                                        FB_Bacnet.StartStopCommand_143.bEnWrite := TRUE;
                                        FB_Bacnet.StartStopCommand_143.bVal := TRUE;
                                    17: 
                                        
                                        FB_Bacnet.StartStopCommand_144.bEnWrite := TRUE;
                                        FB_Bacnet.StartStopCommand_144.bVal := TRUE;
                                    18: 
                                        
                                        FB_Bacnet.StartStopCommand_145.bEnWrite := TRUE;
                                        FB_Bacnet.StartStopCommand_145.bVal := TRUE;
                                    19: 
                                        
                                        FB_Bacnet.StartStopCommand_146.bEnWrite := TRUE;
                                        FB_Bacnet.StartStopCommand_146.bVal := TRUE;
                                    20: 
                                        
                                        FB_Bacnet.StartStopCommand_147.bEnWrite := TRUE;
                                        FB_Bacnet.StartStopCommand_147.bVal := TRUE;
                                    21: 
                                        
                                        FB_Bacnet.StartStopCommand_148.bEnWrite := TRUE;
                                        FB_Bacnet.StartStopCommand_148.bVal := TRUE;
                                    22: 
                                        
                                        FB_Bacnet.StartStopCommand_149.bEnWrite := TRUE;
                                        FB_Bacnet.StartStopCommand_149.bVal := TRUE;
                                    23: 
                                        
                                        FB_Bacnet.StartStopCommand_176.bEnWrite := TRUE;
                                        FB_Bacnet.StartStopCommand_176.bVal := TRUE;
                                    24: 
                                        
                                        FB_Bacnet.StartStopCommand_241.bEnWrite := TRUE;
                                        FB_Bacnet.StartStopCommand_241.bVal := TRUE;
                                    25: 
                                        
                                        FB_Bacnet.StartStopCommand_226.bEnWrite := TRUE;
                                        FB_Bacnet.StartStopCommand_226.bVal := TRUE;
                                END_CASE
                            END_IF
                        END_FOR
                    END_IF
                    // Schedule Unit OFF
                    IF wSchedWDHourEndF38_ = currH AND wSchedWDMinEndF38_ = currM AND NOT bUnitTriggered THEN
                        bUnitTriggered := TRUE;
                        FOR i := 1 TO 25 DO
                            // Send command unit OFF
                            IF bUnitF38_[i] THEN 
                                CASE i OF
                                    1: 
                                        
                                        FB_Bacnet.StartStopCommand_128.bEnWrite := TRUE;
                                        FB_Bacnet.StartStopCommand_128.bVal := FALSE;
                                    2: 
                                        
                                        FB_Bacnet.StartStopCommand_129.bEnWrite := TRUE;
                                        FB_Bacnet.StartStopCommand_129.bVal := FALSE;
                                    3: 
                                        
                                        FB_Bacnet.StartStopCommand_130.bEnWrite := TRUE;
                                        FB_Bacnet.StartStopCommand_130.bVal := FALSE;
                                    4: 
                                        
                                        FB_Bacnet.StartStopCommand_131.bEnWrite := TRUE;
                                        FB_Bacnet.StartStopCommand_131.bVal := FALSE;
                                    5: 
                                        
                                        FB_Bacnet.StartStopCommand_132.bEnWrite := TRUE;
                                        FB_Bacnet.StartStopCommand_132.bVal := FALSE;
                                    6: 
                                        
                                        FB_Bacnet.StartStopCommand_133.bEnWrite := TRUE;
                                        FB_Bacnet.StartStopCommand_133.bVal := FALSE;
                                    7: 
                                        
                                        FB_Bacnet.StartStopCommand_134.bEnWrite := TRUE;
                                        FB_Bacnet.StartStopCommand_134.bVal := FALSE;
                                    8: 
                                        
                                        FB_Bacnet.StartStopCommand_135.bEnWrite := TRUE;
                                        FB_Bacnet.StartStopCommand_135.bVal := FALSE;
                                    9: 
                                        
                                        FB_Bacnet.StartStopCommand_136.bEnWrite := TRUE;
                                        FB_Bacnet.StartStopCommand_136.bVal := FALSE;
                                    10: 
                                        
                                        FB_Bacnet.StartStopCommand_137.bEnWrite := TRUE;
                                        FB_Bacnet.StartStopCommand_137.bVal := FALSE;
                                    11: 
                                        
                                        FB_Bacnet.StartStopCommand_138.bEnWrite := TRUE;
                                        FB_Bacnet.StartStopCommand_138.bVal := FALSE;
                                    12: 
                                        
                                        FB_Bacnet.StartStopCommand_139.bEnWrite := TRUE;
                                        FB_Bacnet.StartStopCommand_139.bVal := FALSE;
                                    13: 
                                        
                                        FB_Bacnet.StartStopCommand_140.bEnWrite := TRUE;
                                        FB_Bacnet.StartStopCommand_140.bVal := FALSE;
                                    14: 
                                        
                                        FB_Bacnet.StartStopCommand_141.bEnWrite := TRUE;
                                        FB_Bacnet.StartStopCommand_141.bVal := FALSE;
                                    15: 
                                        
                                        FB_Bacnet.StartStopCommand_142.bEnWrite := TRUE;
                                        FB_Bacnet.StartStopCommand_142.bVal := FALSE;
                                    16: 
                                        
                                        FB_Bacnet.StartStopCommand_143.bEnWrite := TRUE;
                                        FB_Bacnet.StartStopCommand_143.bVal := FALSE;
                                    17: 
                                        
                                        FB_Bacnet.StartStopCommand_144.bEnWrite := TRUE;
                                        FB_Bacnet.StartStopCommand_144.bVal := FALSE;
                                    18: 
                                        
                                        FB_Bacnet.StartStopCommand_145.bEnWrite := TRUE;
                                        FB_Bacnet.StartStopCommand_145.bVal := FALSE;
                                    19: 
                                        
                                        FB_Bacnet.StartStopCommand_146.bEnWrite := TRUE;
                                        FB_Bacnet.StartStopCommand_146.bVal := FALSE;
                                    20: 
                                        
                                        FB_Bacnet.StartStopCommand_147.bEnWrite := TRUE;
                                        FB_Bacnet.StartStopCommand_147.bVal := FALSE;
                                    21: 
                                        
                                        FB_Bacnet.StartStopCommand_148.bEnWrite := TRUE;
                                        FB_Bacnet.StartStopCommand_148.bVal := FALSE;
                                    22: 
                                        
                                        FB_Bacnet.StartStopCommand_149.bEnWrite := TRUE;
                                        FB_Bacnet.StartStopCommand_149.bVal := FALSE;
                                    23: 
                                        
                                        FB_Bacnet.StartStopCommand_176.bEnWrite := TRUE;
                                        FB_Bacnet.StartStopCommand_176.bVal := FALSE;
                                    24: 
                                        
                                        FB_Bacnet.StartStopCommand_241.bEnWrite := TRUE;
                                        FB_Bacnet.StartStopCommand_241.bVal := FALSE;
                                    25: 
                                        
                                        FB_Bacnet.StartStopCommand_226.bEnWrite := TRUE;
                                        FB_Bacnet.StartStopCommand_226.bVal := FALSE;
                                END_CASE
                            END_IF
                        END_FOR
                    END_IF
                END_IF
            END_IF
        END_IF

        // Weekend schedule
        IF currD = 0 OR currD = 6 THEN
            IF (wSchedWEHourStartF38_ <> wSchedWEHourEndF38_ OR wSchedWEMinStartF38_ <> wSchedWEMinEndF38_) THEN
                // Schedule Unit ON
                IF wSchedWEHourStartF38_ = currH AND wSchedWEMinStartF38_ = currM AND NOT bUnitTriggered THEN
                    bUnitTriggered := TRUE;
                    FOR i := 1 TO 25 DO
                        // Send command unit ON
                        IF bUnitF38_[i] THEN 
                            CASE i OF
                                1: 
                                    
                                    FB_Bacnet.StartStopCommand_128.bEnWrite := TRUE;
                                    FB_Bacnet.StartStopCommand_128.bVal := TRUE;
                                2: 
                                    
                                    FB_Bacnet.StartStopCommand_129.bEnWrite := TRUE;
                                    FB_Bacnet.StartStopCommand_129.bVal := TRUE;
                                3: 
                                    
                                    FB_Bacnet.StartStopCommand_130.bEnWrite := TRUE;
                                    FB_Bacnet.StartStopCommand_130.bVal := TRUE;
                                4: 
                                    
                                    FB_Bacnet.StartStopCommand_131.bEnWrite := TRUE;
                                    FB_Bacnet.StartStopCommand_131.bVal := TRUE;
                                5: 
                                    
                                    FB_Bacnet.StartStopCommand_132.bEnWrite := TRUE;
                                    FB_Bacnet.StartStopCommand_132.bVal := TRUE;
                                6: 
                                    
                                    FB_Bacnet.StartStopCommand_133.bEnWrite := TRUE;
                                    FB_Bacnet.StartStopCommand_133.bVal := TRUE;
                                7: 
                                    
                                    FB_Bacnet.StartStopCommand_134.bEnWrite := TRUE;
                                    FB_Bacnet.StartStopCommand_134.bVal := TRUE;
                                8: 
                                    
                                    FB_Bacnet.StartStopCommand_135.bEnWrite := TRUE;
                                    FB_Bacnet.StartStopCommand_135.bVal := TRUE;
                                9: 
                                    
                                    FB_Bacnet.StartStopCommand_136.bEnWrite := TRUE;
                                    FB_Bacnet.StartStopCommand_136.bVal := TRUE;
                                10: 
                                    
                                    FB_Bacnet.StartStopCommand_137.bEnWrite := TRUE;
                                    FB_Bacnet.StartStopCommand_137.bVal := TRUE;
                                11: 
                                    
                                    FB_Bacnet.StartStopCommand_138.bEnWrite := TRUE;
                                    FB_Bacnet.StartStopCommand_138.bVal := TRUE;
                                12: 
                                    
                                    FB_Bacnet.StartStopCommand_139.bEnWrite := TRUE;
                                    FB_Bacnet.StartStopCommand_139.bVal := TRUE;
                                13: 
                                    
                                    FB_Bacnet.StartStopCommand_140.bEnWrite := TRUE;
                                    FB_Bacnet.StartStopCommand_140.bVal := TRUE;
                                14: 
                                    
                                    FB_Bacnet.StartStopCommand_141.bEnWrite := TRUE;
                                    FB_Bacnet.StartStopCommand_141.bVal := TRUE;
                                15: 
                                    
                                    FB_Bacnet.StartStopCommand_142.bEnWrite := TRUE;
                                    FB_Bacnet.StartStopCommand_142.bVal := TRUE;
                                16: 
                                    
                                    FB_Bacnet.StartStopCommand_143.bEnWrite := TRUE;
                                    FB_Bacnet.StartStopCommand_143.bVal := TRUE;
                                17: 
                                    
                                    FB_Bacnet.StartStopCommand_144.bEnWrite := TRUE;
                                    FB_Bacnet.StartStopCommand_144.bVal := TRUE;
                                18: 
                                    
                                    FB_Bacnet.StartStopCommand_145.bEnWrite := TRUE;
                                    FB_Bacnet.StartStopCommand_145.bVal := TRUE;
                                19: 
                                    
                                    FB_Bacnet.StartStopCommand_146.bEnWrite := TRUE;
                                    FB_Bacnet.StartStopCommand_146.bVal := TRUE;
                                20: 
                                    
                                    FB_Bacnet.StartStopCommand_147.bEnWrite := TRUE;
                                    FB_Bacnet.StartStopCommand_147.bVal := TRUE;
                                21: 
                                    
                                    FB_Bacnet.StartStopCommand_148.bEnWrite := TRUE;
                                    FB_Bacnet.StartStopCommand_148.bVal := TRUE;
                                22: 
                                    
                                    FB_Bacnet.StartStopCommand_149.bEnWrite := TRUE;
                                    FB_Bacnet.StartStopCommand_149.bVal := TRUE;
                                23: 
                                    
                                    FB_Bacnet.StartStopCommand_176.bEnWrite := TRUE;
                                    FB_Bacnet.StartStopCommand_176.bVal := TRUE;
                                24: 
                                    
                                    FB_Bacnet.StartStopCommand_241.bEnWrite := TRUE;
                                    FB_Bacnet.StartStopCommand_241.bVal := TRUE;
                                25: 
                                    
                                    FB_Bacnet.StartStopCommand_226.bEnWrite := TRUE;
                                    FB_Bacnet.StartStopCommand_226.bVal := TRUE;
                            END_CASE
                        END_IF
                    END_FOR        
                END_IF
                // Schedule Unit OFF
                IF wSchedWEHourEndF38_ = currH AND wSchedWEMinEndF38_ = currM AND NOT bUnitTriggered THEN
                    bUnitTriggered := TRUE;
                    FOR i := 1 TO 25 DO
                        // Send command unit OFF
                        IF bUnitF38_[i] THEN 
                            CASE i OF
                                1: 
                                    
                                    FB_Bacnet.StartStopCommand_128.bEnWrite := TRUE;
                                    FB_Bacnet.StartStopCommand_128.bVal := FALSE;
                                2: 
                                    
                                    FB_Bacnet.StartStopCommand_129.bEnWrite := TRUE;
                                    FB_Bacnet.StartStopCommand_129.bVal := FALSE;
                                3: 
                                    
                                    FB_Bacnet.StartStopCommand_130.bEnWrite := TRUE;
                                    FB_Bacnet.StartStopCommand_130.bVal := FALSE;
                                4: 
                                    
                                    FB_Bacnet.StartStopCommand_131.bEnWrite := TRUE;
                                    FB_Bacnet.StartStopCommand_131.bVal := FALSE;
                                5: 
                                    
                                    FB_Bacnet.StartStopCommand_132.bEnWrite := TRUE;
                                    FB_Bacnet.StartStopCommand_132.bVal := FALSE;
                                6: 
                                    
                                    FB_Bacnet.StartStopCommand_133.bEnWrite := TRUE;
                                    FB_Bacnet.StartStopCommand_133.bVal := FALSE;
                                7: 
                                    
                                    FB_Bacnet.StartStopCommand_134.bEnWrite := TRUE;
                                    FB_Bacnet.StartStopCommand_134.bVal := FALSE;
                                8: 
                                    
                                    FB_Bacnet.StartStopCommand_135.bEnWrite := TRUE;
                                    FB_Bacnet.StartStopCommand_135.bVal := FALSE;
                                9: 
                                    
                                    FB_Bacnet.StartStopCommand_136.bEnWrite := TRUE;
                                    FB_Bacnet.StartStopCommand_136.bVal := FALSE;
                                10: 
                                    
                                    FB_Bacnet.StartStopCommand_137.bEnWrite := TRUE;
                                    FB_Bacnet.StartStopCommand_137.bVal := FALSE;
                                11: 
                                    
                                    FB_Bacnet.StartStopCommand_138.bEnWrite := TRUE;
                                    FB_Bacnet.StartStopCommand_138.bVal := FALSE;
                                12: 
                                    
                                    FB_Bacnet.StartStopCommand_139.bEnWrite := TRUE;
                                    FB_Bacnet.StartStopCommand_139.bVal := FALSE;
                                13: 
                                    
                                    FB_Bacnet.StartStopCommand_140.bEnWrite := TRUE;
                                    FB_Bacnet.StartStopCommand_140.bVal := FALSE;
                                14: 
                                    
                                    FB_Bacnet.StartStopCommand_141.bEnWrite := TRUE;
                                    FB_Bacnet.StartStopCommand_141.bVal := FALSE;
                                15: 
                                    
                                    FB_Bacnet.StartStopCommand_142.bEnWrite := TRUE;
                                    FB_Bacnet.StartStopCommand_142.bVal := FALSE;
                                16: 
                                    
                                    FB_Bacnet.StartStopCommand_143.bEnWrite := TRUE;
                                    FB_Bacnet.StartStopCommand_143.bVal := FALSE;
                                17: 
                                    
                                    FB_Bacnet.StartStopCommand_144.bEnWrite := TRUE;
                                    FB_Bacnet.StartStopCommand_144.bVal := FALSE;
                                18: 
                                    
                                    FB_Bacnet.StartStopCommand_145.bEnWrite := TRUE;
                                    FB_Bacnet.StartStopCommand_145.bVal := FALSE;
                                19: 
                                    
                                    FB_Bacnet.StartStopCommand_146.bEnWrite := TRUE;
                                    FB_Bacnet.StartStopCommand_146.bVal := FALSE;
                                20: 
                                    
                                    FB_Bacnet.StartStopCommand_147.bEnWrite := TRUE;
                                    FB_Bacnet.StartStopCommand_147.bVal := FALSE;
                                21: 
                                    
                                    FB_Bacnet.StartStopCommand_148.bEnWrite := TRUE;
                                    FB_Bacnet.StartStopCommand_148.bVal := FALSE;
                                22: 
                                    
                                    FB_Bacnet.StartStopCommand_149.bEnWrite := TRUE;
                                    FB_Bacnet.StartStopCommand_149.bVal := FALSE;
                                23: 
                                    
                                    FB_Bacnet.StartStopCommand_176.bEnWrite := TRUE;
                                    FB_Bacnet.StartStopCommand_176.bVal := FALSE;
                                24: 
                                    
                                    FB_Bacnet.StartStopCommand_241.bEnWrite := TRUE;
                                    FB_Bacnet.StartStopCommand_241.bVal := FALSE;
                                25: 
                                    
                                    FB_Bacnet.StartStopCommand_226.bEnWrite := TRUE;
                                    FB_Bacnet.StartStopCommand_226.bVal := FALSE;
                            END_CASE
                        END_IF
                    END_FOR
                END_IF
            END_IF
        END_IF

END_FUNCTION_BLOCK

// ---- POUs/FB_Scheduler/FB_Scheduler_F39.TcPOU

      FUNCTION_BLOCK FB_Scheduler_F39
      VAR_INPUT
          currH : WORD;
          currM : WORD;
          currD : WORD;
      END_VAR
      VAR_IN_OUT
          FB_Bacnet : FB_BACnet_DAIKIN_MasterStation_III_No_9;
      END_VAR
      VAR
          i : INT;
          prevMinute : WORD := 0;
          bUnitTriggered : BOOL := FALSE;
      END_VAR
      VAR PERSISTENT
          //scheduler var
          bEnSchedF39_ : BOOL := FALSE;
          wSchedWDHourStartF39_ : WORD; 
          wSchedWDMinStartF39_ : WORD; 
          wSchedWEHourStartF39_ : WORD; 
          wSchedWEMinStartF39_ : WORD;
          wSchedWDHourEndF39_ : WORD;
          wSchedWDMinEndF39_ : WORD;
          wSchedWEHourEndF39_ : WORD;
          wSchedWEMinEndF39_ : WORD;
          //unit var
          bUnitF39_ : ARRAY [1..23] OF BOOL;
      END_VAR


        // Reset trigger flag at minute change or at the exact scheduled time
        IF currM <> prevMinute OR 
           (currH = wSchedWDHourStartF39_ AND currM = wSchedWDMinStartF39_) OR 
           (currH = wSchedWDHourEndF39_ AND currM = wSchedWDMinEndF39_) THEN
            bUnitTriggered := FALSE;
            prevMinute := currM;
        END_IF

        // Unit Schedule Enable
        IF bEnSchedF39_ THEN
            // Weekday schedule
            IF currD >= 1 AND currD <= 5 THEN
                IF (wSchedWDHourStartF39_ <> wSchedWDHourEndF39_ OR wSchedWDMinStartF39_ <> wSchedWDMinEndF39_) THEN
                    // Schedule Unit ON
                    IF wSchedWDHourStartF39_ = currH AND wSchedWDMinStartF39_ = currM AND NOT bUnitTriggered THEN
                        bUnitTriggered := TRUE;
                        FOR i := 1 TO 23 DO
                            // Send command unit ON
                            IF bUnitF39_[i] THEN 
                                CASE i OF
                                    1: 
                                        
                                        FB_Bacnet.StartStopCommand_192.bEnWrite := TRUE;
                                        FB_Bacnet.StartStopCommand_192.bVal := TRUE;
                                    2: 
                                        
                                        FB_Bacnet.StartStopCommand_193.bEnWrite := TRUE;
                                        FB_Bacnet.StartStopCommand_193.bVal := TRUE;
                                    3: 
                                        
                                        FB_Bacnet.StartStopCommand_194.bEnWrite := TRUE;
                                        FB_Bacnet.StartStopCommand_194.bVal := TRUE;
                                    4: 
                                        
                                        FB_Bacnet.StartStopCommand_195.bEnWrite := TRUE;
                                        FB_Bacnet.StartStopCommand_195.bVal := TRUE;
                                    5: 
                                        
                                        FB_Bacnet.StartStopCommand_196.bEnWrite := TRUE;
                                        FB_Bacnet.StartStopCommand_196.bVal := TRUE;
                                    6: 
                                        
                                        FB_Bacnet.StartStopCommand_197.bEnWrite := TRUE;
                                        FB_Bacnet.StartStopCommand_197.bVal := TRUE;
                                    7: 
                                        
                                        FB_Bacnet.StartStopCommand_198.bEnWrite := TRUE;
                                        FB_Bacnet.StartStopCommand_198.bVal := TRUE;
                                    8: 
                                        
                                        FB_Bacnet.StartStopCommand_199.bEnWrite := TRUE;
                                        FB_Bacnet.StartStopCommand_199.bVal := TRUE;
                                    9: 
                                        
                                        FB_Bacnet.StartStopCommand_200.bEnWrite := TRUE;
                                        FB_Bacnet.StartStopCommand_200.bVal := TRUE;
                                    10: 
                                        
                                        FB_Bacnet.StartStopCommand_201.bEnWrite := TRUE;
                                        FB_Bacnet.StartStopCommand_201.bVal := TRUE;
                                    11: 
                                        
                                        FB_Bacnet.StartStopCommand_202.bEnWrite := TRUE;
                                        FB_Bacnet.StartStopCommand_202.bVal := TRUE;
                                    12: 
                                        
                                        FB_Bacnet.StartStopCommand_203.bEnWrite := TRUE;
                                        FB_Bacnet.StartStopCommand_203.bVal := TRUE;
                                    13: 
                                        
                                        FB_Bacnet.StartStopCommand_204.bEnWrite := TRUE;
                                        FB_Bacnet.StartStopCommand_204.bVal := TRUE;
                                    14: 
                                        
                                        FB_Bacnet.StartStopCommand_205.bEnWrite := TRUE;
                                        FB_Bacnet.StartStopCommand_205.bVal := TRUE;
                                    15: 
                                        
                                        FB_Bacnet.StartStopCommand_206.bEnWrite := TRUE;
                                        FB_Bacnet.StartStopCommand_206.bVal := TRUE;
                                    16: 
                                        
                                        FB_Bacnet.StartStopCommand_207.bEnWrite := TRUE;
                                        FB_Bacnet.StartStopCommand_207.bVal := TRUE;
                                    17: 
                                        
                                        FB_Bacnet.StartStopCommand_208.bEnWrite := TRUE;
                                        FB_Bacnet.StartStopCommand_208.bVal := TRUE;
                                    18: 
                                        
                                        FB_Bacnet.StartStopCommand_209.bEnWrite := TRUE;
                                        FB_Bacnet.StartStopCommand_209.bVal := TRUE;
                                    19: 
                                        
                                        FB_Bacnet.StartStopCommand_210.bEnWrite := TRUE;
                                        FB_Bacnet.StartStopCommand_210.bVal := TRUE;
                                    20: 
                                        
                                        FB_Bacnet.StartStopCommand_211.bEnWrite := TRUE;
                                        FB_Bacnet.StartStopCommand_211.bVal := TRUE;
                                    21: 
                                        
                                        FB_Bacnet.StartStopCommand_212.bEnWrite := TRUE;
                                        FB_Bacnet.StartStopCommand_212.bVal := TRUE;
                                    22: 
                                        
                                        FB_Bacnet.StartStopCommand_213.bEnWrite := TRUE;
                                        FB_Bacnet.StartStopCommand_213.bVal := TRUE;
                                    23: 
                                        
                                        FB_Bacnet.StartStopCommand_227.bEnWrite := TRUE;
                                        FB_Bacnet.StartStopCommand_227.bVal := TRUE;
                                END_CASE
                            END_IF
                        END_FOR
                    END_IF
                    // Schedule Unit OFF
                    IF wSchedWDHourEndF39_ = currH AND wSchedWDMinEndF39_ = currM AND NOT bUnitTriggered THEN
                        bUnitTriggered := TRUE;
                        FOR i := 1 TO 23 DO
                            // Send command unit OFF
                            IF bUnitF39_[i] THEN 
                                CASE i OF
                                    1: 
                                        
                                        FB_Bacnet.StartStopCommand_192.bEnWrite := TRUE;
                                        FB_Bacnet.StartStopCommand_192.bVal := FALSE;
                                    2: 
                                        
                                        FB_Bacnet.StartStopCommand_193.bEnWrite := TRUE;
                                        FB_Bacnet.StartStopCommand_193.bVal := FALSE;
                                    3: 
                                        
                                        FB_Bacnet.StartStopCommand_194.bEnWrite := TRUE;
                                        FB_Bacnet.StartStopCommand_194.bVal := FALSE;
                                    4: 
                                        
                                        FB_Bacnet.StartStopCommand_195.bEnWrite := TRUE;
                                        FB_Bacnet.StartStopCommand_195.bVal := FALSE;
                                    5: 
                                        
                                        FB_Bacnet.StartStopCommand_196.bEnWrite := TRUE;
                                        FB_Bacnet.StartStopCommand_196.bVal := FALSE;
                                    6: 
                                        
                                        FB_Bacnet.StartStopCommand_197.bEnWrite := TRUE;
                                        FB_Bacnet.StartStopCommand_197.bVal := FALSE;
                                    7: 
                                        
                                        FB_Bacnet.StartStopCommand_198.bEnWrite := TRUE;
                                        FB_Bacnet.StartStopCommand_198.bVal := FALSE;
                                    8: 
                                        
                                        FB_Bacnet.StartStopCommand_199.bEnWrite := TRUE;
                                        FB_Bacnet.StartStopCommand_199.bVal := FALSE;
                                    9: 
                                        
                                        FB_Bacnet.StartStopCommand_200.bEnWrite := TRUE;
                                        FB_Bacnet.StartStopCommand_200.bVal := FALSE;
                                    10: 
                                        
                                        FB_Bacnet.StartStopCommand_201.bEnWrite := TRUE;
                                        FB_Bacnet.StartStopCommand_201.bVal := FALSE;
                                    11: 
                                        
                                        FB_Bacnet.StartStopCommand_202.bEnWrite := TRUE;
                                        FB_Bacnet.StartStopCommand_202.bVal := FALSE;
                                    12: 
                                        
                                        FB_Bacnet.StartStopCommand_203.bEnWrite := TRUE;
                                        FB_Bacnet.StartStopCommand_203.bVal := FALSE;
                                    13: 
                                        
                                        FB_Bacnet.StartStopCommand_204.bEnWrite := TRUE;
                                        FB_Bacnet.StartStopCommand_204.bVal := FALSE;
                                    14: 
                                        
                                        FB_Bacnet.StartStopCommand_205.bEnWrite := TRUE;
                                        FB_Bacnet.StartStopCommand_205.bVal := FALSE;
                                    15: 
                                        
                                        FB_Bacnet.StartStopCommand_206.bEnWrite := TRUE;
                                        FB_Bacnet.StartStopCommand_206.bVal := FALSE;
                                    16: 
                                        
                                        FB_Bacnet.StartStopCommand_207.bEnWrite := TRUE;
                                        FB_Bacnet.StartStopCommand_207.bVal := FALSE;
                                    17: 
                                        
                                        FB_Bacnet.StartStopCommand_208.bEnWrite := TRUE;
                                        FB_Bacnet.StartStopCommand_208.bVal := FALSE;
                                    18: 
                                        
                                        FB_Bacnet.StartStopCommand_209.bEnWrite := TRUE;
                                        FB_Bacnet.StartStopCommand_209.bVal := FALSE;
                                    19: 
                                        
                                        FB_Bacnet.StartStopCommand_210.bEnWrite := TRUE;
                                        FB_Bacnet.StartStopCommand_210.bVal := FALSE;
                                    20: 
                                        
                                        FB_Bacnet.StartStopCommand_211.bEnWrite := TRUE;
                                        FB_Bacnet.StartStopCommand_211.bVal := FALSE;
                                    21: 
                                        
                                        FB_Bacnet.StartStopCommand_212.bEnWrite := TRUE;
                                        FB_Bacnet.StartStopCommand_212.bVal := FALSE;
                                    22: 
                                        
                                        FB_Bacnet.StartStopCommand_213.bEnWrite := TRUE;
                                        FB_Bacnet.StartStopCommand_213.bVal := FALSE;
                                    23: 
                                        
                                        FB_Bacnet.StartStopCommand_227.bEnWrite := TRUE;
                                        FB_Bacnet.StartStopCommand_227.bVal := FALSE;
                                END_CASE
                            END_IF
                        END_FOR
                    END_IF
                END_IF
            END_IF

            // Weekend schedule
            IF currD = 0 OR currD = 6 THEN
                IF (wSchedWEHourStartF39_ <> wSchedWEHourEndF39_ OR wSchedWEMinStartF39_ <> wSchedWEMinEndF39_) THEN
                    // Schedule Unit ON
                    IF wSchedWEHourStartF39_ = currH AND wSchedWEMinStartF39_ = currM AND NOT bUnitTriggered THEN
                        bUnitTriggered := TRUE;
                        FOR i := 1 TO 23 DO
                            // Send command unit ON
                            IF bUnitF39_[i] THEN 
                                CASE i OF
                                    1: 
                                        
                                        FB_Bacnet.StartStopCommand_192.bEnWrite := TRUE;
                                        FB_Bacnet.StartStopCommand_192.bVal := TRUE;
                                    2: 
                                        
                                        FB_Bacnet.StartStopCommand_193.bEnWrite := TRUE;
                                        FB_Bacnet.StartStopCommand_193.bVal := TRUE;
                                    3: 
                                        
                                        FB_Bacnet.StartStopCommand_194.bEnWrite := TRUE;
                                        FB_Bacnet.StartStopCommand_194.bVal := TRUE;
                                    4: 
                                        
                                        FB_Bacnet.StartStopCommand_195.bEnWrite := TRUE;
                                        FB_Bacnet.StartStopCommand_195.bVal := TRUE;
                                    5: 
                                        
                                        FB_Bacnet.StartStopCommand_196.bEnWrite := TRUE;
                                        FB_Bacnet.StartStopCommand_196.bVal := TRUE;
                                    6: 
                                        
                                        FB_Bacnet.StartStopCommand_197.bEnWrite := TRUE;
                                        FB_Bacnet.StartStopCommand_197.bVal := TRUE;
                                    7: 
                                        
                                        FB_Bacnet.StartStopCommand_198.bEnWrite := TRUE;
                                        FB_Bacnet.StartStopCommand_198.bVal := TRUE;
                                    8: 
                                        
                                        FB_Bacnet.StartStopCommand_199.bEnWrite := TRUE;
                                        FB_Bacnet.StartStopCommand_199.bVal := TRUE;
                                    9: 
                                        
                                        FB_Bacnet.StartStopCommand_200.bEnWrite := TRUE;
                                        FB_Bacnet.StartStopCommand_200.bVal := TRUE;
                                    10: 
                                        
                                        FB_Bacnet.StartStopCommand_201.bEnWrite := TRUE;
                                        FB_Bacnet.StartStopCommand_201.bVal := TRUE;
                                    11: 
                                        
                                        FB_Bacnet.StartStopCommand_202.bEnWrite := TRUE;
                                        FB_Bacnet.StartStopCommand_202.bVal := TRUE;
                                    12: 
                                        
                                        FB_Bacnet.StartStopCommand_203.bEnWrite := TRUE;
                                        FB_Bacnet.StartStopCommand_203.bVal := TRUE;
                                    13: 
                                        
                                        FB_Bacnet.StartStopCommand_204.bEnWrite := TRUE;
                                        FB_Bacnet.StartStopCommand_204.bVal := TRUE;
                                    14: 
                                        
                                        FB_Bacnet.StartStopCommand_205.bEnWrite := TRUE;
                                        FB_Bacnet.StartStopCommand_205.bVal := TRUE;
                                    15: 
                                        
                                        FB_Bacnet.StartStopCommand_206.bEnWrite := TRUE;
                                        FB_Bacnet.StartStopCommand_206.bVal := TRUE;
                                    16: 
                                        
                                        FB_Bacnet.StartStopCommand_207.bEnWrite := TRUE;
                                        FB_Bacnet.StartStopCommand_207.bVal := TRUE;
                                    17: 
                                        
                                        FB_Bacnet.StartStopCommand_208.bEnWrite := TRUE;
                                        FB_Bacnet.StartStopCommand_208.bVal := TRUE;
                                    18: 
                                        
                                        FB_Bacnet.StartStopCommand_209.bEnWrite := TRUE;
                                        FB_Bacnet.StartStopCommand_209.bVal := TRUE;
                                    19: 
                                        
                                        FB_Bacnet.StartStopCommand_210.bEnWrite := TRUE;
                                        FB_Bacnet.StartStopCommand_210.bVal := TRUE;
                                    20: 
                                        
                                        FB_Bacnet.StartStopCommand_211.bEnWrite := TRUE;
                                        FB_Bacnet.StartStopCommand_211.bVal := TRUE;
                                    21: 
                                        
                                        FB_Bacnet.StartStopCommand_212.bEnWrite := TRUE;
                                        FB_Bacnet.StartStopCommand_212.bVal := TRUE;
                                    22: 
                                        
                                        FB_Bacnet.StartStopCommand_213.bEnWrite := TRUE;
                                        FB_Bacnet.StartStopCommand_213.bVal := TRUE;
                                    23: 
                                        
                                        FB_Bacnet.StartStopCommand_227.bEnWrite := TRUE;
                                        FB_Bacnet.StartStopCommand_227.bVal := TRUE;
                                END_CASE
                            END_IF
                        END_FOR
                    END_IF
                    // Schedule Unit OFF
                    IF wSchedWEHourEndF39_ = currH AND wSchedWEMinEndF39_ = currM AND NOT bUnitTriggered THEN
                        bUnitTriggered := TRUE;
                        FOR i := 1 TO 23 DO
                            // Send command unit OFF
                            IF bUnitF39_[i] THEN 
                                CASE i OF
                                    1: 
                                        
                                        FB_Bacnet.StartStopCommand_192.bEnWrite := TRUE;
                                        FB_Bacnet.StartStopCommand_192.bVal := FALSE;
                                    2: 
                                        
                                        FB_Bacnet.StartStopCommand_193.bEnWrite := TRUE;
                                        FB_Bacnet.StartStopCommand_193.bVal := FALSE;
                                    3: 
                                        
                                        FB_Bacnet.StartStopCommand_194.bEnWrite := TRUE;
                                        FB_Bacnet.StartStopCommand_194.bVal := FALSE;
                                    4: 
                                        
                                        FB_Bacnet.StartStopCommand_195.bEnWrite := TRUE;
                                        FB_Bacnet.StartStopCommand_195.bVal := FALSE;
                                    5: 
                                        
                                        FB_Bacnet.StartStopCommand_196.bEnWrite := TRUE;
                                        FB_Bacnet.StartStopCommand_196.bVal := FALSE;
                                    6: 
                                        
                                        FB_Bacnet.StartStopCommand_197.bEnWrite := TRUE;
                                        FB_Bacnet.StartStopCommand_197.bVal := FALSE;
                                    7: 
                                        
                                        FB_Bacnet.StartStopCommand_198.bEnWrite := TRUE;
                                        FB_Bacnet.StartStopCommand_198.bVal := FALSE;
                                    8: 
                                        
                                        FB_Bacnet.StartStopCommand_199.bEnWrite := TRUE;
                                        FB_Bacnet.StartStopCommand_199.bVal := FALSE;
                                    9: 
                                        
                                        FB_Bacnet.StartStopCommand_200.bEnWrite := TRUE;
                                        FB_Bacnet.StartStopCommand_200.bVal := FALSE;
                                    10: 
                                        
                                        FB_Bacnet.StartStopCommand_201.bEnWrite := TRUE;
                                        FB_Bacnet.StartStopCommand_201.bVal := FALSE;
                                    11: 
                                        
                                        FB_Bacnet.StartStopCommand_202.bEnWrite := TRUE;
                                        FB_Bacnet.StartStopCommand_202.bVal := FALSE;
                                    12: 
                                        
                                        FB_Bacnet.StartStopCommand_203.bEnWrite := TRUE;
                                        FB_Bacnet.StartStopCommand_203.bVal := FALSE;
                                    13: 
                                        
                                        FB_Bacnet.StartStopCommand_204.bEnWrite := TRUE;
                                        FB_Bacnet.StartStopCommand_204.bVal := FALSE;
                                    14: 
                                        
                                        FB_Bacnet.StartStopCommand_205.bEnWrite := TRUE;
                                        FB_Bacnet.StartStopCommand_205.bVal := FALSE;
                                    15: 
                                        
                                        FB_Bacnet.StartStopCommand_206.bEnWrite := TRUE;
                                        FB_Bacnet.StartStopCommand_206.bVal := FALSE;
                                    16: 
                                        
                                        FB_Bacnet.StartStopCommand_207.bEnWrite := TRUE;
                                        FB_Bacnet.StartStopCommand_207.bVal := FALSE;
                                    17: 
                                        
                                        FB_Bacnet.StartStopCommand_208.bEnWrite := TRUE;
                                        FB_Bacnet.StartStopCommand_208.bVal := FALSE;
                                    18: 
                                        
                                        FB_Bacnet.StartStopCommand_209.bEnWrite := TRUE;
                                        FB_Bacnet.StartStopCommand_209.bVal := FALSE;
                                    19: 
                                        
                                        FB_Bacnet.StartStopCommand_210.bEnWrite := TRUE;
                                        FB_Bacnet.StartStopCommand_210.bVal := FALSE;
                                    20: 
                                        
                                        FB_Bacnet.StartStopCommand_211.bEnWrite := TRUE;
                                        FB_Bacnet.StartStopCommand_211.bVal := FALSE;
                                    21: 
                                        
                                        FB_Bacnet.StartStopCommand_212.bEnWrite := TRUE;
                                        FB_Bacnet.StartStopCommand_212.bVal := FALSE;
                                    22: 
                                        
                                        FB_Bacnet.StartStopCommand_213.bEnWrite := TRUE;
                                        FB_Bacnet.StartStopCommand_213.bVal := FALSE;
                                    23: 
                                        
                                        FB_Bacnet.StartStopCommand_227.bEnWrite := TRUE;
                                        FB_Bacnet.StartStopCommand_227.bVal := FALSE;
                                END_CASE
                            END_IF
                        END_FOR
                    END_IF
                END_IF
            END_IF
        END_IF

END_FUNCTION_BLOCK

// ---- POUs/FB_Scheduler/FB_Scheduler_F50.TcPOU

      FUNCTION_BLOCK FB_Scheduler_F50
      VAR_INPUT
          currH : WORD;
          currM : WORD;
          currD : WORD;
      END_VAR
      VAR_IN_OUT
          FB_Bacnet : FB_BACnet_DAIKIN_MasterStation_III_No_10;
      END_VAR
      VAR
          i : INT;
          bUnitTriggered : BOOL := FALSE; // New flag to track execution
          prevMinute : WORD := 0;        // New variable to track the previous minute
      END_VAR
      VAR PERSISTENT
          //scheduler var
          bEnSchedF50_ : BOOL := FALSE;
          wSchedWDHourStartF50_ : WORD; 
          wSchedWDMinStartF50_ : WORD; 
          wSchedWEHourStartF50_ : WORD; 
          wSchedWEMinStartF50_ : WORD;
          wSchedWDHourEndF50_ : WORD;
          wSchedWDMinEndF50_ : WORD;
          wSchedWEHourEndF50_ : WORD;
          wSchedWEMinEndF50_ : WORD;
          //unit var
          bUnitF50_ : ARRAY [1..23] OF BOOL;
      END_VAR


        // Reset trigger flag at minute change or at the exact scheduled time
        IF currM <> prevMinute OR 
           (currH = wSchedWDHourStartF50_ AND currM = wSchedWDMinStartF50_) OR 
           (currH = wSchedWDHourEndF50_ AND currM = wSchedWDMinEndF50_) THEN
            bUnitTriggered := FALSE;
            prevMinute := currM;
        END_IF

        // Unit Schedule Enable
        IF bEnSchedF50_ THEN
            // Weekday schedule
            IF currD >= 1 AND currD <= 5 THEN
                IF (wSchedWDHourStartF50_ <> wSchedWDHourEndF50_ OR wSchedWDMinStartF50_ <> wSchedWDMinEndF50_) THEN
                    // Schedule Unit ON
                    IF wSchedWDHourStartF50_ = currH AND wSchedWDMinStartF50_ = currM AND NOT bUnitTriggered THEN
                        bUnitTriggered := TRUE;
                        FOR i := 1 TO 23 DO
                            // Send command unit ON
                            IF bUnitF50_[i] THEN 
                                CASE i OF
                                    1: 
                                        
                                        FB_Bacnet.StartStopCommand_000.bEnWrite := TRUE;
                                        FB_Bacnet.StartStopCommand_000.bVal := TRUE;
                                    2: 
                                        
                                        FB_Bacnet.StartStopCommand_001.bEnWrite := TRUE;
                                        FB_Bacnet.StartStopCommand_001.bVal := TRUE;
                                    3: 
                                        
                                        FB_Bacnet.StartStopCommand_002.bEnWrite := TRUE;
                                        FB_Bacnet.StartStopCommand_002.bVal := TRUE;
                                    4: 
                                        
                                        FB_Bacnet.StartStopCommand_003.bEnWrite := TRUE;
                                        FB_Bacnet.StartStopCommand_003.bVal := TRUE;
                                    5: 
                                        
                                        FB_Bacnet.StartStopCommand_004.bEnWrite := TRUE;
                                        FB_Bacnet.StartStopCommand_004.bVal := TRUE;
                                    6: 
                                        
                                        FB_Bacnet.StartStopCommand_005.bEnWrite := TRUE;
                                        FB_Bacnet.StartStopCommand_005.bVal := TRUE;
                                    7: 
                                        
                                        FB_Bacnet.StartStopCommand_006.bEnWrite := TRUE;
                                        FB_Bacnet.StartStopCommand_006.bVal := TRUE;
                                    8: 
                                        
                                        FB_Bacnet.StartStopCommand_007.bEnWrite := TRUE;
                                        FB_Bacnet.StartStopCommand_007.bVal := TRUE;
                                    9: 
                                        
                                        FB_Bacnet.StartStopCommand_008.bEnWrite := TRUE;
                                        FB_Bacnet.StartStopCommand_008.bVal := TRUE;
                                    10: 
                                        
                                        FB_Bacnet.StartStopCommand_009.bEnWrite := TRUE;
                                        FB_Bacnet.StartStopCommand_009.bVal := TRUE;
                                    11: 
                                        
                                        FB_Bacnet.StartStopCommand_010.bEnWrite := TRUE;
                                        FB_Bacnet.StartStopCommand_010.bVal := TRUE;
                                    12: 
                                        
                                        FB_Bacnet.StartStopCommand_011.bEnWrite := TRUE;
                                        FB_Bacnet.StartStopCommand_011.bVal := TRUE;
                                    13: 
                                        
                                        FB_Bacnet.StartStopCommand_012.bEnWrite := TRUE;
                                        FB_Bacnet.StartStopCommand_012.bVal := TRUE;
                                    14: 
                                        
                                        FB_Bacnet.StartStopCommand_013.bEnWrite := TRUE;
                                        FB_Bacnet.StartStopCommand_013.bVal := TRUE;
                                    15: 
                                        
                                        FB_Bacnet.StartStopCommand_014.bEnWrite := TRUE;
                                        FB_Bacnet.StartStopCommand_014.bVal := TRUE;
                                    16: 
                                        
                                        FB_Bacnet.StartStopCommand_015.bEnWrite := TRUE;
                                        FB_Bacnet.StartStopCommand_015.bVal := TRUE;
                                    17: 
                                        
                                        FB_Bacnet.StartStopCommand_016.bEnWrite := TRUE;
                                        FB_Bacnet.StartStopCommand_016.bVal := TRUE;
                                    18: 
                                        
                                        FB_Bacnet.StartStopCommand_017.bEnWrite := TRUE;
                                        FB_Bacnet.StartStopCommand_017.bVal := TRUE;
                                    19: 
                                        
                                        FB_Bacnet.StartStopCommand_018.bEnWrite := TRUE;
                                        FB_Bacnet.StartStopCommand_018.bVal := TRUE;
                                    20: 
                                        
                                        FB_Bacnet.StartStopCommand_019.bEnWrite := TRUE;
                                        FB_Bacnet.StartStopCommand_019.bVal := TRUE;
                                    21: 
                                        
                                        FB_Bacnet.StartStopCommand_020.bEnWrite := TRUE;
                                        FB_Bacnet.StartStopCommand_020.bVal := TRUE;
                                    22: 
                                        
                                        FB_Bacnet.StartStopCommand_021.bEnWrite := TRUE;
                                        FB_Bacnet.StartStopCommand_021.bVal := TRUE;
                                    23: 
                                        
                                        FB_Bacnet.StartStopCommand_234.bEnWrite := TRUE;
                                        FB_Bacnet.StartStopCommand_234.bVal := TRUE;
                                END_CASE
                            END_IF
                        END_FOR
                    END_IF
                    // Schedule Unit OFF
                    IF wSchedWDHourEndF50_ = currH AND wSchedWDMinEndF50_ = currM AND NOT bUnitTriggered THEN
                        bUnitTriggered := TRUE;
                        FOR i := 1 TO 23 DO
                            // Send command unit OFF
                            IF bUnitF50_[i] THEN 
                                CASE i OF
                                    1: 
                                        
                                        FB_Bacnet.StartStopCommand_000.bEnWrite := TRUE;
                                        FB_Bacnet.StartStopCommand_000.bVal := FALSE;
                                    2: 
                                        
                                        FB_Bacnet.StartStopCommand_001.bEnWrite := TRUE;
                                        FB_Bacnet.StartStopCommand_001.bVal := FALSE;
                                    3: 
                                        
                                        FB_Bacnet.StartStopCommand_002.bEnWrite := TRUE;
                                        FB_Bacnet.StartStopCommand_002.bVal := FALSE;
                                    4: 
                                        
                                        FB_Bacnet.StartStopCommand_003.bEnWrite := TRUE;
                                        FB_Bacnet.StartStopCommand_003.bVal := FALSE;
                                    5: 
                                        
                                        FB_Bacnet.StartStopCommand_004.bEnWrite := TRUE;
                                        FB_Bacnet.StartStopCommand_004.bVal := FALSE;
                                    6: 
                                        
                                        FB_Bacnet.StartStopCommand_005.bEnWrite := TRUE;
                                        FB_Bacnet.StartStopCommand_005.bVal := FALSE;
                                    7: 
                                        
                                        FB_Bacnet.StartStopCommand_006.bEnWrite := TRUE;
                                        FB_Bacnet.StartStopCommand_006.bVal := FALSE;
                                    8: 
                                        
                                        FB_Bacnet.StartStopCommand_007.bEnWrite := TRUE;
                                        FB_Bacnet.StartStopCommand_007.bVal := FALSE;
                                    9: 
                                        
                                        FB_Bacnet.StartStopCommand_008.bEnWrite := TRUE;
                                        FB_Bacnet.StartStopCommand_008.bVal := FALSE;
                                    10: 
                                        
                                        FB_Bacnet.StartStopCommand_009.bEnWrite := TRUE;
                                        FB_Bacnet.StartStopCommand_009.bVal := FALSE;
                                    11: 
                                        
                                        FB_Bacnet.StartStopCommand_010.bEnWrite := TRUE;
                                        FB_Bacnet.StartStopCommand_010.bVal := FALSE;
                                    12: 
                                        
                                        FB_Bacnet.StartStopCommand_011.bEnWrite := TRUE;
                                        FB_Bacnet.StartStopCommand_011.bVal := FALSE;
                                    13: 
                                        
                                        FB_Bacnet.StartStopCommand_012.bEnWrite := TRUE;
                                        FB_Bacnet.StartStopCommand_012.bVal := FALSE;
                                    14: 
                                        
                                        FB_Bacnet.StartStopCommand_013.bEnWrite := TRUE;
                                        FB_Bacnet.StartStopCommand_013.bVal := FALSE;
                                    15: 
                                        
                                        FB_Bacnet.StartStopCommand_014.bEnWrite := TRUE;
                                        FB_Bacnet.StartStopCommand_014.bVal := FALSE;
                                    16: 
                                        
                                        FB_Bacnet.StartStopCommand_015.bEnWrite := TRUE;
                                        FB_Bacnet.StartStopCommand_015.bVal := FALSE;
                                    17: 
                                        
                                        FB_Bacnet.StartStopCommand_016.bEnWrite := TRUE;
                                        FB_Bacnet.StartStopCommand_016.bVal := FALSE;
                                    18: 
                                        
                                        FB_Bacnet.StartStopCommand_017.bEnWrite := TRUE;
                                        FB_Bacnet.StartStopCommand_017.bVal := FALSE;
                                    19: 
                                        
                                        FB_Bacnet.StartStopCommand_018.bEnWrite := TRUE;
                                        FB_Bacnet.StartStopCommand_018.bVal := FALSE;
                                    20: 
                                        
                                        FB_Bacnet.StartStopCommand_019.bEnWrite := TRUE;
                                        FB_Bacnet.StartStopCommand_019.bVal := FALSE;
                                    21: 
                                        
                                        FB_Bacnet.StartStopCommand_020.bEnWrite := TRUE;
                                        FB_Bacnet.StartStopCommand_020.bVal := FALSE;
                                    22: 
                                        
                                        FB_Bacnet.StartStopCommand_021.bEnWrite := TRUE;
                                        FB_Bacnet.StartStopCommand_021.bVal := FALSE;
                                    23: 
                                        
                                        FB_Bacnet.StartStopCommand_234.bEnWrite := TRUE;
                                        FB_Bacnet.StartStopCommand_234.bVal := FALSE;
                                END_CASE
                            END_IF
                        END_FOR
                    END_IF
                END_IF
            END_IF

            // Weekend schedule
            IF currD = 0 OR currD = 6 THEN
                IF (wSchedWEHourStartF50_ <> wSchedWEHourEndF50_ OR wSchedWEMinStartF50_ <> wSchedWEMinEndF50_) THEN
                    // Schedule Unit ON
                    IF wSchedWEHourStartF50_ = currH AND wSchedWEMinStartF50_ = currM AND NOT bUnitTriggered THEN
                        bUnitTriggered := TRUE;
                        FOR i := 1 TO 23 DO
                            // Send command unit ON
                            IF bUnitF50_[i] THEN 
                                CASE i OF
                                    1: 
                                        
                                        FB_Bacnet.StartStopCommand_000.bEnWrite := TRUE;
                                        FB_Bacnet.StartStopCommand_000.bVal := TRUE;
                                    2: 
                                        
                                        FB_Bacnet.StartStopCommand_001.bEnWrite := TRUE;
                                        FB_Bacnet.StartStopCommand_001.bVal := TRUE;
                                    3: 
                                        
                                        FB_Bacnet.StartStopCommand_002.bEnWrite := TRUE;
                                        FB_Bacnet.StartStopCommand_002.bVal := TRUE;
                                    4: 
                                        
                                        FB_Bacnet.StartStopCommand_003.bEnWrite := TRUE;
                                        FB_Bacnet.StartStopCommand_003.bVal := TRUE;
                                    5: 
                                        
                                        FB_Bacnet.StartStopCommand_004.bEnWrite := TRUE;
                                        FB_Bacnet.StartStopCommand_004.bVal := TRUE;
                                    6: 
                                        
                                        FB_Bacnet.StartStopCommand_005.bEnWrite := TRUE;
                                        FB_Bacnet.StartStopCommand_005.bVal := TRUE;
                                    7: 
                                        
                                        FB_Bacnet.StartStopCommand_006.bEnWrite := TRUE;
                                        FB_Bacnet.StartStopCommand_006.bVal := TRUE;
                                    8: 
                                        
                                        FB_Bacnet.StartStopCommand_007.bEnWrite := TRUE;
                                        FB_Bacnet.StartStopCommand_007.bVal := TRUE;
                                    9: 
                                        
                                        FB_Bacnet.StartStopCommand_008.bEnWrite := TRUE;
                                        FB_Bacnet.StartStopCommand_008.bVal := TRUE;
                                    10: 
                                        
                                        FB_Bacnet.StartStopCommand_009.bEnWrite := TRUE;
                                        FB_Bacnet.StartStopCommand_009.bVal := TRUE;
                                    11: 
                                        
                                        FB_Bacnet.StartStopCommand_010.bEnWrite := TRUE;
                                        FB_Bacnet.StartStopCommand_010.bVal := TRUE;
                                    12: 
                                        
                                        FB_Bacnet.StartStopCommand_011.bEnWrite := TRUE;
                                        FB_Bacnet.StartStopCommand_011.bVal := TRUE;
                                    13: 
                                        
                                        FB_Bacnet.StartStopCommand_012.bEnWrite := TRUE;
                                        FB_Bacnet.StartStopCommand_012.bVal := TRUE;
                                    14: 
                                        
                                        FB_Bacnet.StartStopCommand_013.bEnWrite := TRUE;
                                        FB_Bacnet.StartStopCommand_013.bVal := TRUE;
                                    15: 
                                        
                                        FB_Bacnet.StartStopCommand_014.bEnWrite := TRUE;
                                        FB_Bacnet.StartStopCommand_014.bVal := TRUE;
                                    16: 
                                        
                                        FB_Bacnet.StartStopCommand_015.bEnWrite := TRUE;
                                        FB_Bacnet.StartStopCommand_015.bVal := TRUE;
                                    17: 
                                        
                                        FB_Bacnet.StartStopCommand_016.bEnWrite := TRUE;
                                        FB_Bacnet.StartStopCommand_016.bVal := TRUE;
                                    18: 
                                        
                                        FB_Bacnet.StartStopCommand_017.bEnWrite := TRUE;
                                        FB_Bacnet.StartStopCommand_017.bVal := TRUE;
                                    19: 
                                        
                                        FB_Bacnet.StartStopCommand_018.bEnWrite := TRUE;
                                        FB_Bacnet.StartStopCommand_018.bVal := TRUE;
                                    20: 
                                        
                                        FB_Bacnet.StartStopCommand_019.bEnWrite := TRUE;
                                        FB_Bacnet.StartStopCommand_019.bVal := TRUE;
                                    21: 
                                        
                                        FB_Bacnet.StartStopCommand_020.bEnWrite := TRUE;
                                        FB_Bacnet.StartStopCommand_020.bVal := TRUE;
                                    22: 
                                        
                                        FB_Bacnet.StartStopCommand_021.bEnWrite := TRUE;
                                        FB_Bacnet.StartStopCommand_021.bVal := TRUE;
                                    23: 
                                        
                                        FB_Bacnet.StartStopCommand_234.bEnWrite := TRUE;
                                        FB_Bacnet.StartStopCommand_234.bVal := TRUE;
                                END_CASE
                            END_IF
                        END_FOR
                    END_IF
                    // Schedule Unit OFF
                    IF wSchedWEHourEndF50_ = currH AND wSchedWEMinEndF50_ = currM AND NOT bUnitTriggered THEN
                        bUnitTriggered := TRUE;
                        FOR i := 1 TO 23 DO
                            // Send command unit OFF
                            IF bUnitF50_[i] THEN 
                                CASE i OF
                                    1: 
                                        
                                        FB_Bacnet.StartStopCommand_000.bEnWrite := TRUE;
                                        FB_Bacnet.StartStopCommand_000.bVal := FALSE;
                                    2: 
                                        
                                        FB_Bacnet.StartStopCommand_001.bEnWrite := TRUE;
                                        FB_Bacnet.StartStopCommand_001.bVal := FALSE;
                                    3: 
                                        
                                        FB_Bacnet.StartStopCommand_002.bEnWrite := TRUE;
                                        FB_Bacnet.StartStopCommand_002.bVal := FALSE;
                                    4: 
                                        
                                        FB_Bacnet.StartStopCommand_003.bEnWrite := TRUE;
                                        FB_Bacnet.StartStopCommand_003.bVal := FALSE;
                                    5: 
                                        
                                        FB_Bacnet.StartStopCommand_004.bEnWrite := TRUE;
                                        FB_Bacnet.StartStopCommand_004.bVal := FALSE;
                                    6: 
                                        
                                        FB_Bacnet.StartStopCommand_005.bEnWrite := TRUE;
                                        FB_Bacnet.StartStopCommand_005.bVal := FALSE;
                                    7: 
                                        
                                        FB_Bacnet.StartStopCommand_006.bEnWrite := TRUE;
                                        FB_Bacnet.StartStopCommand_006.bVal := FALSE;
                                    8: 
                                        
                                        FB_Bacnet.StartStopCommand_007.bEnWrite := TRUE;
                                        FB_Bacnet.StartStopCommand_007.bVal := FALSE;
                                    9: 
                                        
                                        FB_Bacnet.StartStopCommand_008.bEnWrite := TRUE;
                                        FB_Bacnet.StartStopCommand_008.bVal := FALSE;
                                    10: 
                                        
                                        FB_Bacnet.StartStopCommand_009.bEnWrite := TRUE;
                                        FB_Bacnet.StartStopCommand_009.bVal := FALSE;
                                    11: 
                                        
                                        FB_Bacnet.StartStopCommand_010.bEnWrite := TRUE;
                                        FB_Bacnet.StartStopCommand_010.bVal := FALSE;
                                    12: 
                                        
                                        FB_Bacnet.StartStopCommand_011.bEnWrite := TRUE;
                                        FB_Bacnet.StartStopCommand_011.bVal := FALSE;
                                    13: 
                                        
                                        FB_Bacnet.StartStopCommand_012.bEnWrite := TRUE;
                                        FB_Bacnet.StartStopCommand_012.bVal := FALSE;
                                    14: 
                                        
                                        FB_Bacnet.StartStopCommand_013.bEnWrite := TRUE;
                                        FB_Bacnet.StartStopCommand_013.bVal := FALSE;
                                    15: 
                                        
                                        FB_Bacnet.StartStopCommand_014.bEnWrite := TRUE;
                                        FB_Bacnet.StartStopCommand_014.bVal := FALSE;
                                    16: 
                                        
                                        FB_Bacnet.StartStopCommand_015.bEnWrite := TRUE;
                                        FB_Bacnet.StartStopCommand_015.bVal := FALSE;
                                    17: 
                                        
                                        FB_Bacnet.StartStopCommand_016.bEnWrite := TRUE;
                                        FB_Bacnet.StartStopCommand_016.bVal := FALSE;
                                    18: 
                                        
                                        FB_Bacnet.StartStopCommand_017.bEnWrite := TRUE;
                                        FB_Bacnet.StartStopCommand_017.bVal := FALSE;
                                    19: 
                                        
                                        FB_Bacnet.StartStopCommand_018.bEnWrite := TRUE;
                                        FB_Bacnet.StartStopCommand_018.bVal := FALSE;
                                    20: 
                                        
                                        FB_Bacnet.StartStopCommand_019.bEnWrite := TRUE;
                                        FB_Bacnet.StartStopCommand_019.bVal := FALSE;
                                    21: 
                                        
                                        FB_Bacnet.StartStopCommand_020.bEnWrite := TRUE;
                                        FB_Bacnet.StartStopCommand_020.bVal := FALSE;
                                    22: 
                                        
                                        FB_Bacnet.StartStopCommand_021.bEnWrite := TRUE;
                                        FB_Bacnet.StartStopCommand_021.bVal := FALSE;
                                    23: 
                                        
                                        FB_Bacnet.StartStopCommand_234.bEnWrite := TRUE;
                                        FB_Bacnet.StartStopCommand_234.bVal := FALSE;
                                END_CASE
                            END_IF
                        END_FOR
                    END_IF
                END_IF
            END_IF
        END_IF

END_FUNCTION_BLOCK

// ---- POUs/FB_Scheduler/FB_Scheduler_F51.TcPOU

      FUNCTION_BLOCK FB_Scheduler_F51
      VAR_INPUT
          currH : WORD;
          currM : WORD;
          currD : WORD;
      END_VAR
      VAR_IN_OUT
          FB_Bacnet : FB_BACnet_DAIKIN_MasterStation_III_No_10;
      END_VAR
      VAR
          i : INT;
          bUnitTriggered : BOOL := FALSE; // New flag to track execution
          prevMinute : WORD := 0;        // New variable to track the previous minute
      END_VAR
      VAR PERSISTENT
          //scheduler var
          bEnSchedF51_ : BOOL := FALSE;
          wSchedWDHourStartF51_ : WORD; 
          wSchedWDMinStartF51_ : WORD; 
          wSchedWEHourStartF51_ : WORD; 
          wSchedWEMinStartF51_ : WORD;
          wSchedWDHourEndF51_ : WORD;
          wSchedWDMinEndF51_ : WORD;
          wSchedWEHourEndF51_ : WORD;
          wSchedWEMinEndF51_ : WORD;
          //unit var
          bUnitF51_ : ARRAY [1..25] OF BOOL;
      END_VAR


// Reset trigger flag at minute change or at the exact scheduled time
IF currM <> prevMinute OR 
   (currH = wSchedWDHourStartF51_ AND currM = wSchedWDMinStartF51_) OR 
   (currH = wSchedWDHourEndF51_ AND currM = wSchedWDMinEndF51_) THEN
    bUnitTriggered := FALSE;
    prevMinute := currM;
END_IF

// Unit Schedule Enable
IF bEnSchedF51_ THEN
    // Weekday schedule
    IF currD >= 1 AND currD <= 5 THEN
        IF (wSchedWDHourStartF51_ <> wSchedWDHourEndF51_ OR wSchedWDMinStartF51_ <> wSchedWDMinEndF51_) THEN
            // Schedule Unit ON
            IF wSchedWDHourStartF51_ = currH AND wSchedWDMinStartF51_ = currM AND NOT bUnitTriggered THEN
                bUnitTriggered := TRUE;
                FOR i := 1 TO 25 DO
                    //send command unit ON
                    IF bUnitF51_[i] = TRUE THEN 
                        CASE i OF
                            1: 
                                
                                FB_Bacnet.StartStopCommand_064.bEnWrite := TRUE;
                                FB_Bacnet.StartStopCommand_064.bVal := TRUE;
                            2: 
                                
                                FB_Bacnet.StartStopCommand_065.bEnWrite := TRUE;
                                FB_Bacnet.StartStopCommand_065.bVal := TRUE;
                            3: 
                                
                                FB_Bacnet.StartStopCommand_066.bEnWrite := TRUE;
                                FB_Bacnet.StartStopCommand_066.bVal := TRUE;
                            4: 
                                
                                FB_Bacnet.StartStopCommand_067.bEnWrite := TRUE;
                                FB_Bacnet.StartStopCommand_067.bVal := TRUE;
                            5: 
                                
                                FB_Bacnet.StartStopCommand_068.bEnWrite := TRUE;
                                FB_Bacnet.StartStopCommand_068.bVal := TRUE;
                            6: 
                                
                                FB_Bacnet.StartStopCommand_069.bEnWrite := TRUE;
                                FB_Bacnet.StartStopCommand_069.bVal := TRUE;
                            7: 
                                
                                FB_Bacnet.StartStopCommand_070.bEnWrite := TRUE;
                                FB_Bacnet.StartStopCommand_070.bVal := TRUE;
                            8: 
                                
                                FB_Bacnet.StartStopCommand_071.bEnWrite := TRUE;
                                FB_Bacnet.StartStopCommand_071.bVal := TRUE;
                            9: 
                                
                                FB_Bacnet.StartStopCommand_072.bEnWrite := TRUE;
                                FB_Bacnet.StartStopCommand_072.bVal := TRUE;
                            10: 
                                
                                FB_Bacnet.StartStopCommand_073.bEnWrite := TRUE;
                                FB_Bacnet.StartStopCommand_073.bVal := TRUE;
                            11: 
                                
                                FB_Bacnet.StartStopCommand_074.bEnWrite := TRUE;
                                FB_Bacnet.StartStopCommand_074.bVal := TRUE;
                            12: 
                                
                                FB_Bacnet.StartStopCommand_075.bEnWrite := TRUE;
                                FB_Bacnet.StartStopCommand_075.bVal := TRUE;
                            13: 
                                
                                FB_Bacnet.StartStopCommand_076.bEnWrite := TRUE;
                                FB_Bacnet.StartStopCommand_076.bVal := TRUE;
                            14: 
                                
                                FB_Bacnet.StartStopCommand_077.bEnWrite := TRUE;
                                FB_Bacnet.StartStopCommand_077.bVal := TRUE;
                            15: 
                                
                                FB_Bacnet.StartStopCommand_078.bEnWrite := TRUE;
                                FB_Bacnet.StartStopCommand_078.bVal := TRUE;
                            16: 
                                
                                FB_Bacnet.StartStopCommand_079.bEnWrite := TRUE;
                                FB_Bacnet.StartStopCommand_079.bVal := TRUE;
                            17: 
                                
                                FB_Bacnet.StartStopCommand_080.bEnWrite := TRUE;
                                FB_Bacnet.StartStopCommand_080.bVal := TRUE;
                            18: 
                                
                                FB_Bacnet.StartStopCommand_081.bEnWrite := TRUE;
                                FB_Bacnet.StartStopCommand_081.bVal := TRUE;
                            19: 
                                
                                FB_Bacnet.StartStopCommand_082.bEnWrite := TRUE;
                                FB_Bacnet.StartStopCommand_082.bVal := TRUE;
                            20: 
                                
                                FB_Bacnet.StartStopCommand_083.bEnWrite := TRUE;
                                FB_Bacnet.StartStopCommand_083.bVal := TRUE;
                            21: 
                                
                                FB_Bacnet.StartStopCommand_084.bEnWrite := TRUE;
                                FB_Bacnet.StartStopCommand_084.bVal := TRUE;
                            22: 
                                
                                FB_Bacnet.StartStopCommand_085.bEnWrite := TRUE;
                                FB_Bacnet.StartStopCommand_085.bVal := TRUE;
                            23: 
                                
                                FB_Bacnet.StartStopCommand_112.bEnWrite := TRUE;
                                FB_Bacnet.StartStopCommand_112.bVal := TRUE;
                            24: 
                                
                                FB_Bacnet.StartStopCommand_241.bEnWrite := TRUE;
                                FB_Bacnet.StartStopCommand_241.bVal := TRUE;
                            25: 
                                
                                FB_Bacnet.StartStopCommand_235.bEnWrite := TRUE;
                                FB_Bacnet.StartStopCommand_235.bVal := TRUE;
                        END_CASE
                    END_IF
                END_FOR
            END_IF
            // Schedule Unit OFF
            IF wSchedWDHourEndF51_ = currH AND wSchedWDMinEndF51_ = currM AND NOT bUnitTriggered THEN
                bUnitTriggered := TRUE;
                FOR i := 1 TO 25 DO
                    //send command unit OFF
                    IF bUnitF51_[i] = TRUE THEN 
                        CASE i OF
                            1: 
                                
                                FB_Bacnet.StartStopCommand_064.bEnWrite := TRUE;
                                FB_Bacnet.StartStopCommand_064.bVal := FALSE;
                            2: 
                                
                                FB_Bacnet.StartStopCommand_065.bEnWrite := TRUE;
                                FB_Bacnet.StartStopCommand_065.bVal := FALSE;
                            3: 
                                
                                FB_Bacnet.StartStopCommand_066.bEnWrite := TRUE;
                                FB_Bacnet.StartStopCommand_066.bVal := FALSE;
                            4: 
                                
                                FB_Bacnet.StartStopCommand_067.bEnWrite := TRUE;
                                FB_Bacnet.StartStopCommand_067.bVal := FALSE;
                            5: 
                                
                                FB_Bacnet.StartStopCommand_068.bEnWrite := TRUE;
                                FB_Bacnet.StartStopCommand_068.bVal := FALSE;
                            6: 
                                
                                FB_Bacnet.StartStopCommand_069.bEnWrite := TRUE;
                                FB_Bacnet.StartStopCommand_069.bVal := FALSE;
                            7: 
                                
                                FB_Bacnet.StartStopCommand_070.bEnWrite := TRUE;
                                FB_Bacnet.StartStopCommand_070.bVal := FALSE;
                            8: 
                                
                                FB_Bacnet.StartStopCommand_071.bEnWrite := TRUE;
                                FB_Bacnet.StartStopCommand_071.bVal := FALSE;
                            9: 
                                
                                FB_Bacnet.StartStopCommand_072.bEnWrite := TRUE;
                                FB_Bacnet.StartStopCommand_072.bVal := FALSE;
                            10: 
                                
                                FB_Bacnet.StartStopCommand_073.bEnWrite := TRUE;
                                FB_Bacnet.StartStopCommand_073.bVal := FALSE;
                            11: 
                                
                                FB_Bacnet.StartStopCommand_074.bEnWrite := TRUE;
                                FB_Bacnet.StartStopCommand_074.bVal := FALSE;
                            12: 
                                
                                FB_Bacnet.StartStopCommand_075.bEnWrite := TRUE;
                                FB_Bacnet.StartStopCommand_075.bVal := FALSE;
                            13: 
                                
                                FB_Bacnet.StartStopCommand_076.bEnWrite := TRUE;
                                FB_Bacnet.StartStopCommand_076.bVal := FALSE;
                            14: 
                                
                                FB_Bacnet.StartStopCommand_077.bEnWrite := TRUE;
                                FB_Bacnet.StartStopCommand_077.bVal := FALSE;
                            15: 
                                
                                FB_Bacnet.StartStopCommand_078.bEnWrite := TRUE;
                                FB_Bacnet.StartStopCommand_078.bVal := FALSE;
                            16: 
                                
                                FB_Bacnet.StartStopCommand_079.bEnWrite := TRUE;
                                FB_Bacnet.StartStopCommand_079.bVal := FALSE;
                            17: 
                                
                                FB_Bacnet.StartStopCommand_080.bEnWrite := TRUE;
                                FB_Bacnet.StartStopCommand_080.bVal := FALSE;
                            18: 
                                
                                FB_Bacnet.StartStopCommand_081.bEnWrite := TRUE;
                                FB_Bacnet.StartStopCommand_081.bVal := FALSE;
                            19: 
                                
                                FB_Bacnet.StartStopCommand_082.bEnWrite := TRUE;
                                FB_Bacnet.StartStopCommand_082.bVal := FALSE;
                            20: 
                                
                                FB_Bacnet.StartStopCommand_083.bEnWrite := TRUE;
                                FB_Bacnet.StartStopCommand_083.bVal := FALSE;
                            21: 
                                
                                FB_Bacnet.StartStopCommand_084.bEnWrite := TRUE;
                                FB_Bacnet.StartStopCommand_084.bVal := FALSE;
                            22: 
                                
                                FB_Bacnet.StartStopCommand_085.bEnWrite := TRUE;
                                FB_Bacnet.StartStopCommand_085.bVal := FALSE;
                            23: 
                                
                                FB_Bacnet.StartStopCommand_112.bEnWrite := TRUE;
                                FB_Bacnet.StartStopCommand_112.bVal := FALSE;
                            24: 
                                
                                FB_Bacnet.StartStopCommand_241.bEnWrite := TRUE;
                                FB_Bacnet.StartStopCommand_241.bVal := FALSE;
                            25: 
                                
                                FB_Bacnet.StartStopCommand_235.bEnWrite := TRUE;
                                FB_Bacnet.StartStopCommand_235.bVal := FALSE;
                        END_CASE
                    END_IF
                END_FOR
            END_IF
        END_IF
    END_IF

    // Weekend schedule
    IF currD = 0 OR currD = 6 THEN
        IF (wSchedWEHourStartF51_ <> wSchedWEHourEndF51_ OR wSchedWEMinStartF51_ <> wSchedWEMinEndF51_) THEN
            // Schedule Unit ON
            IF wSchedWEHourStartF51_ = currH AND wSchedWEMinStartF51_ = currM AND NOT bUnitTriggered THEN
                bUnitTriggered := TRUE;
                FOR i := 1 TO 25 DO
                    //send command unit ON
                    IF bUnitF51_[i] = TRUE THEN 
                        CASE i OF
                            1: 
                                
                                FB_Bacnet.StartStopCommand_064.bEnWrite := TRUE;
                                FB_Bacnet.StartStopCommand_064.bVal := TRUE;
                            2: 
                                
                                FB_Bacnet.StartStopCommand_065.bEnWrite := TRUE;
                                FB_Bacnet.StartStopCommand_065.bVal := TRUE;
                            3: 
                                
                                FB_Bacnet.StartStopCommand_066.bEnWrite := TRUE;
                                FB_Bacnet.StartStopCommand_066.bVal := TRUE;
                            4: 
                                
                                FB_Bacnet.StartStopCommand_067.bEnWrite := TRUE;
                                FB_Bacnet.StartStopCommand_067.bVal := TRUE;
                            5: 
                                
                                FB_Bacnet.StartStopCommand_068.bEnWrite := TRUE;
                                FB_Bacnet.StartStopCommand_068.bVal := TRUE;
                            6: 
                                
                                FB_Bacnet.StartStopCommand_069.bEnWrite := TRUE;
                                FB_Bacnet.StartStopCommand_069.bVal := TRUE;
                            7: 
                                
                                FB_Bacnet.StartStopCommand_070.bEnWrite := TRUE;
                                FB_Bacnet.StartStopCommand_070.bVal := TRUE;
                            8: 
                                
                                FB_Bacnet.StartStopCommand_071.bEnWrite := TRUE;
                                FB_Bacnet.StartStopCommand_071.bVal := TRUE;
                            9: 
                                
                                FB_Bacnet.StartStopCommand_072.bEnWrite := TRUE;
                                FB_Bacnet.StartStopCommand_072.bVal := TRUE;
                            10: 
                                
                                FB_Bacnet.StartStopCommand_073.bEnWrite := TRUE;
                                FB_Bacnet.StartStopCommand_073.bVal := TRUE;
                            11: 
                                
                                FB_Bacnet.StartStopCommand_074.bEnWrite := TRUE;
                                FB_Bacnet.StartStopCommand_074.bVal := TRUE;
                            12: 
                                
                                FB_Bacnet.StartStopCommand_075.bEnWrite := TRUE;
                                FB_Bacnet.StartStopCommand_075.bVal := TRUE;
                            13: 
                                
                                FB_Bacnet.StartStopCommand_076.bEnWrite := TRUE;
                                FB_Bacnet.StartStopCommand_076.bVal := TRUE;
                            14: 
                                
                                FB_Bacnet.StartStopCommand_077.bEnWrite := TRUE;
                                FB_Bacnet.StartStopCommand_077.bVal := TRUE;
                            15: 
                                
                                FB_Bacnet.StartStopCommand_078.bEnWrite := TRUE;
                                FB_Bacnet.StartStopCommand_078.bVal := TRUE;
                            16: 
                                
                                FB_Bacnet.StartStopCommand_079.bEnWrite := TRUE;
                                FB_Bacnet.StartStopCommand_079.bVal := TRUE;
                            17: 
                                
                                FB_Bacnet.StartStopCommand_080.bEnWrite := TRUE;
                                FB_Bacnet.StartStopCommand_080.bVal := TRUE;
                            18: 
                                
                                FB_Bacnet.StartStopCommand_081.bEnWrite := TRUE;
                                FB_Bacnet.StartStopCommand_081.bVal := TRUE;
                            19: 
                                
                                FB_Bacnet.StartStopCommand_082.bEnWrite := TRUE;
                                FB_Bacnet.StartStopCommand_082.bVal := TRUE;
                            20: 
                                
                                FB_Bacnet.StartStopCommand_083.bEnWrite := TRUE;
                                FB_Bacnet.StartStopCommand_083.bVal := TRUE;
                            21: 
                                
                                FB_Bacnet.StartStopCommand_084.bEnWrite := TRUE;
                                FB_Bacnet.StartStopCommand_084.bVal := TRUE;
                            22: 
                                
                                FB_Bacnet.StartStopCommand_085.bEnWrite := TRUE;
                                FB_Bacnet.StartStopCommand_085.bVal := TRUE;
                            23: 
                                
                                FB_Bacnet.StartStopCommand_112.bEnWrite := TRUE;
                                FB_Bacnet.StartStopCommand_112.bVal := TRUE;
                            24: 
                                
                                FB_Bacnet.StartStopCommand_241.bEnWrite := TRUE;
                                FB_Bacnet.StartStopCommand_241.bVal := TRUE;
                            25: 
                                
                                FB_Bacnet.StartStopCommand_235.bEnWrite := TRUE;
                                FB_Bacnet.StartStopCommand_235.bVal := TRUE;
                        END_CASE
                    END_IF
                END_FOR        
            END_IF
            // Schedule Unit OFF
            IF wSchedWEHourEndF51_ = currH AND wSchedWEMinEndF51_ = currM AND NOT bUnitTriggered THEN
                bUnitTriggered := TRUE;
                FOR i := 1 TO 25 DO
                    //send command unit OFF
                    IF bUnitF51_[i] = TRUE THEN 
                        CASE i OF
                            1: 
                                
                                FB_Bacnet.StartStopCommand_064.bEnWrite := TRUE;
                                FB_Bacnet.StartStopCommand_064.bVal := FALSE;
                            2: 
                                
                                FB_Bacnet.StartStopCommand_065.bEnWrite := TRUE;
                                FB_Bacnet.StartStopCommand_065.bVal := FALSE;
                            3: 
                                
                                FB_Bacnet.StartStopCommand_066.bEnWrite := TRUE;
                                FB_Bacnet.StartStopCommand_066.bVal := FALSE;
                            4: 
                                
                                FB_Bacnet.StartStopCommand_067.bEnWrite := TRUE;
                                FB_Bacnet.StartStopCommand_067.bVal := FALSE;
                            5: 
                                
                                FB_Bacnet.StartStopCommand_068.bEnWrite := TRUE;
                                FB_Bacnet.StartStopCommand_068.bVal := FALSE;
                            6: 
                                
                                FB_Bacnet.StartStopCommand_069.bEnWrite := TRUE;
                                FB_Bacnet.StartStopCommand_069.bVal := FALSE;
                            7: 
                                
                                FB_Bacnet.StartStopCommand_070.bEnWrite := TRUE;
                                FB_Bacnet.StartStopCommand_070.bVal := FALSE;
                            8: 
                                
                                FB_Bacnet.StartStopCommand_071.bEnWrite := TRUE;
                                FB_Bacnet.StartStopCommand_071.bVal := FALSE;
                            9: 
                                
